Staubli VAL3: onInsert.pgx

public program onInsert(string& x_sItem[])
  local num l_nSize
  local num i
  local num l_nKey
  local string l_sMessage
  local string l_sItem
  local bool l_bActive
  local num l_nIndex
  local string l_sType
  local num l_nSizeList
  local num l_nValue
  local string l_sName
  local string l_sItemList
begin
  cls()
  x_sItem=""
  call getSize(l_nSizeList)
  l_nSize=0
  //
  // create the list
  //
  call use:setSizeList(10,0,28,11)
  call use:listcreate("OUTPUT ")
  // insert in the list
  for i=0 to l_nSizeList-1
    call out:get(l_sItem,i)
    call out:isActive(l_bActive,l_sItem)
    if l_bActive
      // insert into the list
      call out:getItem(l_sName,l_sItem)
      l_sItemList=l_sItem+" {"+l_sName+"}"
      call use:listadd(l_sItemList)
    endIf
  endFor
  call use:listredraw(min(l_nIndex-use:nView,0))
  // display the actual item
  call getType(l_sType)
  l_sItem=l_sType
  call use:clear(0,13)
  call language:message(l_sMessage,63)
  call use:typeCenter(13,l_sMessage,40,false)
  do
    l_nKey=get()
    // get one output from the list
    call use:listevent(l_nKey,l_nIndex,l_sItem)
    if l_nKey==255
      return
    endIf
  until l_nKey==270
  // insert the pulse
  call use:insertDialog("DELAY [Sec] ",l_nValue,0,100)
  if !use:bUseEscape
    //
    // insert the sentence
    //
    if l_sItem==""
      return
    else
      l_sItem=left(l_sItem,find(l_sItem,"{")-1)
    endIf
    // return the value
    x_sItem="OUT "+l_sItem+">ON,"+toString(".2",l_nValue)
  endIf
end
